(* IEC 61131-3 sources: Industry-PLC-LLM/data/PLCBEAD_repo/PLCBEAD_PLCEmbed-main/PLC-BEAD/Source/GEB/SECOND, 1 file *)

(* ---- SECOND.ST ---- *)
FUNCTION SECOND:REAL

	VAR_INPUT
		ITOD :	UDINT;
	END_VAR

	second := UDINT_TO_REAL(itod MOD UDINT#60000) / REAL#1000.00;

END_FUNCTION

PROGRAM program0
  VAR
    ITOD :	UDINT;
    CEIL5_OUT : REAL;
  END_VAR

  CEIL5_OUT := SECOND(ITOD);
END_PROGRAM
